{attribute 'enable_dynamic_creation'}
FUNCTION_BLOCK ABSTRACT FB_Helper
VAR
END_VAR

// Helper implementation

METHOD PUBLIC ImportConfigFromFile : BOOL
VAR_INPUT
	sFilePath : STRING(255);
END_VAR
// TODO: Implement file import
END_METHOD

METHOD PUBLIC LoadFrameConfigFromFile : BOOL
VAR_INPUT
	sFilePath : STRING(255);
END_VAR
// TODO: Implement frame config load
END_METHOD

METHOD PUBLIC LoadTargetConfigFromFile : BOOL
VAR_INPUT
	sFilePath : STRING(255);
END_VAR
// TODO: Implement target config load
END_METHOD

METHOD PUBLIC LoadToolConfigFromFile : BOOL
VAR_INPUT
	sFilePath : STRING(255);
END_VAR
// TODO: Implement tool config load
END_METHOD

METHOD PUBLIC SaveConfigToFile : BOOL
VAR_INPUT
	sFilePath : STRING(255);
END_VAR
// TODO: Implement file save
END_METHOD

METHOD PUBLIC SaveFrameConfigToFile : BOOL
VAR_INPUT
	sFilePath : STRING(255);
END_VAR
// TODO: Implement frame config save
END_METHOD

METHOD PUBLIC SaveTargetConfigToFile : BOOL
VAR_INPUT
	sFilePath : STRING(255);
END_VAR
// TODO: Implement target config save
END_METHOD

METHOD PUBLIC SaveToolConfigToFile : BOOL
VAR_INPUT
	sFilePath : STRING(255);
END_VAR
// TODO: Implement tool config save
END_METHOD

END_FUNCTION_BLOCK

(* stored: Version 1.1.0.1, ProductVersion 3.1.4026.18
   POU FB_Helper: Id {e1b2c3d4-1111-1111-1111-111111111111}, SpecialFunc None
   Method ImportConfigFromFile: Id {e1b2c3d4-1121-1111-1111-111111111111}
   Method LoadFrameConfigFromFile: Id {e1b2c3d4-1124-1111-1111-111111111111}
   Method LoadTargetConfigFromFile: Id {e1b2c3d4-1125-1111-1111-111111111111}
   Method LoadToolConfigFromFile: Id {e1b2c3d4-1123-1111-1111-111111111111}
   Method SaveConfigToFile: Id {e1b2c3d4-1122-1111-1111-111111111111}
   Method SaveFrameConfigToFile: Id {e1b2c3d4-1127-1111-1111-111111111111}
   Method SaveTargetConfigToFile: Id {e1b2c3d4-1128-1111-1111-111111111111}
   Method SaveToolConfigToFile: Id {e1b2c3d4-1126-1111-1111-111111111111} *)
